// TIA Portal V18 export
// export: Created 2026-06-20T23:26:23.319602Z, ExportSetting WithDefaults
TextList "TL_Mixing_Step"  ListRange=Decimal, Comment="Mã bước chu trình Mixing"
  TextListEntry   EntryType=SingleValue, Text="Chờ lệnh"
  TextListEntry   EntryType=SingleValue, From=10, To=10, Text="Dosing nước"
  TextListEntry   EntryType=SingleValue, From=11, To=11, Text="Tip nguyên liệu"
  TextListEntry   EntryType=SingleValue, From=12, To=12, Text="Khuấy ban đầu"
  TextListEntry   EntryType=SingleValue, From=15, To=15, Text="Xả sang bồn kế tiếp"
  TextListEntry   EntryType=SingleValue, From=20, To=20, Text="Dosing bổ sung"
  TextListEntry   EntryType=SingleValue, From=21, To=21, Text="Tip phụ gia"
  TextListEntry   EntryType=SingleValue, From=22, To=22, Text="Khuấy chiều thuận"
  TextListEntry   EntryType=SingleValue, From=23, To=23, Text="Khuấy chiều ngược"
  TextListEntry   EntryType=SingleValue, From=30, To=30, Text="PID gia nhiệt/điều khiển"
  TextListEntry   EntryType=SingleValue, From=31, To=31, Text="Giữ thanh trùng"
  TextListEntry   EntryType=SingleValue, From=50, To=50, Text="Bồn chứa 01 nhận dịch"
  TextListEntry   EntryType=SingleValue, From=60, To=60, Text="Giải nhiệt"
  TextListEntry   EntryType=SingleValue, From=70, To=70, Text="Chuyển sang Bồn chứa 02"
  TextListEntry   EntryType=SingleValue, From=80, To=80, Text="Lọc CCP và chiết rót"
